ABB RobotStudio station: Robotstudio-car-assembly.rspag

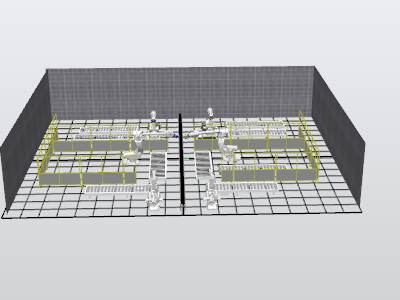
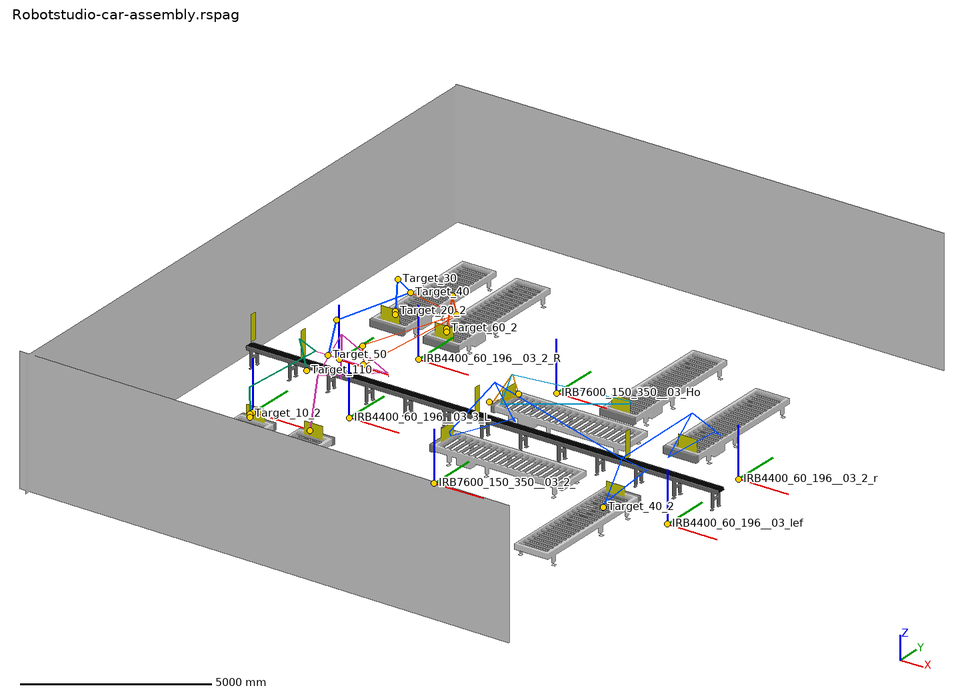
[picture v1: parts stored in the station drawn from their meshes, with robot base, taught points and paths (robot models come from the ABB library and are not in the file)]
--- station ---
Station Project_re_RS (saved by RobotStudio 25.3.11371.0)
Controller Controller29, task T_ROB2: task frame (RAPID world) sits at (6953.35, -1606.5, 0) mm, rotated rx 0 ry 0 rz 180 deg in the station
Controller Controller29, task T_ROB1: task frame (RAPID world) sits at (6953.35, -1606.5, 0) mm, rotated rx 0 ry 0 rz 180 deg in the station
Controller Controller25, task T_ROB2: task frame (RAPID world) sits at (641.16, 3478.05, 0) mm, rotated rx 0 ry 0 rz -90 deg in the station
Controller Controller25, task T_ROB1: task frame (RAPID world) sits at (641.16, 3478.05, 0) mm, rotated rx 0 ry 0 rz -90 deg in the station
Controller Controller23, task T_ROB2: task frame (RAPID world) sits at (-5299.47, 2064.24, 374.5) mm in the station
Controller Controller23, task T_ROB1: task frame (RAPID world) sits at (-5299.47, 2064.24, 374.5) mm in the station
Controller Controller23
  mechanical unit ROB_1: IRB4400_60_196__03_2_Right_Wheel, 6 joints, base frame (0, 0, 0) mm
  mechanical unit TRACK_1: IRBT4004_STD_0_0_3__04_RightWheel, 1 joints, base frame (0, 0, 0) mm
  mechanical unit ROB_2: IRB4400_60_196__03_3_Left_Wheel, 6 joints, base frame (0, 0, 0) mm
  mechanical unit TRACK_2: IRBT4004_STD_0_0_3__04_2_LeftWheel, 1 joints, base frame (-36.16, -3878.12, 0) mm
Controller Controller25
  mechanical unit ROB_1: IRB7600_150_350__03_HoodWind, 6 joints, base frame (358.26, -535.69, 0) mm
  mechanical unit ROB_2: IRB7600_150_350__03_2_Seat, 6 joints, base frame (6589.94, -77.42, 0) mm, rotated rx 0 ry 0 rz 180 deg
Controller Controller29
  mechanical unit ROB_1: IRB4400_60_196__03_leftSide, 6 joints, base frame (0, 0, 0) mm
  mechanical unit ROB_2: IRB4400_60_196__03_2_rightSide, 6 joints, base frame (15.31, -3252.7, 0) mm
Layout (positions relative to the parent item):
  - SmartComponent_Kaross [smart component]
      signals: DI diStartBelt, DI diNewStation, DO doStartBelt, DO dosink, DI diSink
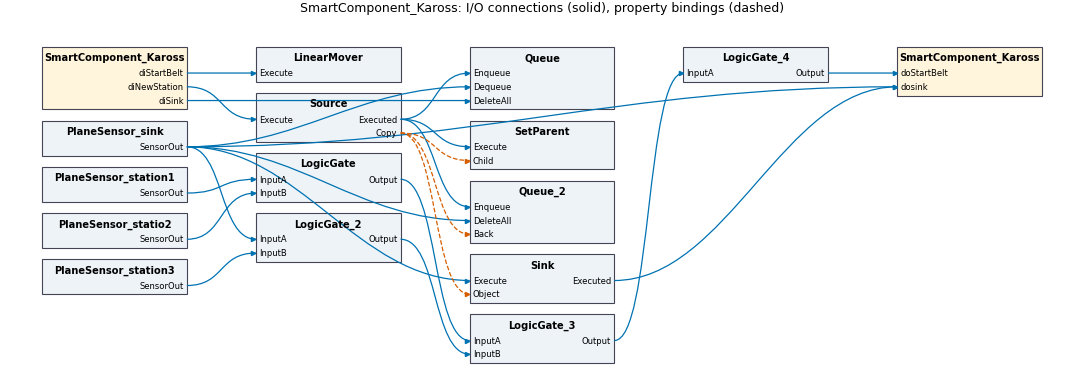
      connections:
        SmartComponent_Kaross.diStartBelt -> LinearMover.Execute
        Source.Executed -> Queue.Enqueue
        PlaneSensor_sink.SensorOut -> Sink.Execute
        PlaneSensor_sink.SensorOut -> Queue.Dequeue
        Source.Executed -> SetParent.Execute
        PlaneSensor_station1.SensorOut -> LogicGate.InputA
        PlaneSensor_statio2.SensorOut -> LogicGate.InputB
        PlaneSensor_sink.SensorOut -> LogicGate_2.InputA
        PlaneSensor_station3.SensorOut -> LogicGate_2.InputB
        LogicGate.Output -> LogicGate_3.InputA
        LogicGate_2.Output -> LogicGate_3.InputB
        LogicGate_3.Output -> LogicGate_4.InputA
        LogicGate_4.Output -> SmartComponent_Kaross.doStartBelt
        SmartComponent_Kaross.diNewStation -> Source.Execute
        Sink.Executed -> SmartComponent_Kaross.dosink
        SmartComponent_Kaross.diSink -> Queue.DeleteAll
        Source.Executed -> Queue_2.Enqueue
        PlaneSensor_sink.SensorOut -> Queue_2.DeleteAll
        PlaneSensor_sink.SensorOut -> SmartComponent_Kaross.dosink
        Source.Copy => SetParent.Child
        Source.Copy => Sink.Object
        Source.Copy => Queue_2.Back
    - Belt Conveyor [part], size 15091 x 400 x 600 mm
    - kaross [part], size 2040 x 1220 x 356.4 mm
    - Source [smart component, from Components\Source.rslib]
        properties: Source=kaross; Copy=(none); Parent=(none); Position=[0 0 0]; Orientation=[0 0 0]; Transient=false; PhysicsBehavior=-1
    - Queue [smart component, from Components\Queue.rslib]
        properties: Back=CAR; Front=(none); Queue=; NumberOfObjects=0
    - LinearMover [smart component, from Components\LinearMover.rslib]
        properties: Object=Queue; Direction=[-1 0 0]; Speed=0.5; Reference=Global; ReferenceObject=(none)
    - PlaneSensor_station1 [smart component, from Components\PlaneSensor.rslib] at (4530.08, -56.57, 1401.52) mm, rotated rx -90 ry 0 rz 90 deg
        properties: Origin=[0 0 0]; Axis1=[0.2 0 0]; Axis2=[0 0.8 0]; Tag=(none); SenseMultiple=false; SensedPart=(none)
      - _sensorPart_ [part], size 200 x 800 x 0 mm
    - PlaneSensor_sink [smart component, from Components\PlaneSensor.rslib] at (-7451.46, 0, 1424.26) mm, rotated rx -90 ry 0 rz 90 deg
        properties: Origin=[0 0 0]; Axis1=[0.2 0 0]; Axis2=[0 0.8 0]; Tag=(none); SenseMultiple=false; SensedPart=(none)
      - _sensorPart_ [part], size 200 x 800 x 0 mm
    - PlaneSensor_statio2 [smart component, from Components\PlaneSensor.rslib] at (-173.15, 0, 622.02) mm, rotated rx 90 ry 0 rz -90 deg
        properties: Origin=[0 0 0]; Axis1=[0.2 0 0]; Axis2=[0 0.8 0]; Tag=(none); SenseMultiple=false; SensedPart=(none)
      - _sensorPart_ [part], size 200 x 800 x 0 mm
    - PlaneSensor_station3 [smart component, from Components\PlaneSensor.rslib] at (-5859.99, 0, 1399.15) mm, rotated rx -90 ry 0 rz 90 deg
        properties: Origin=[0 0 0]; Axis1=[0.2 0 0]; Axis2=[0 0.8 0]; Tag=(none); SenseMultiple=false; SensedPart=(none)
      - _sensorPart_ [part], size 200 x 800 x 0 mm
    - SetParent [smart component, from Components\SetParent.rslib]
        properties: Child=(none); Parent=CAR; KeepTransform=true
    - LogicGate [smart component, from Components\LogicGate.rslib]
        properties: Operator=OR; Delay=0
    - LogicGate_2 [smart component, from Components\LogicGate.rslib]
        properties: Operator=OR; Delay=0
    - LogicGate_3 [smart component, from Components\LogicGate.rslib]
        properties: Operator=OR; Delay=0
    - LogicGate_4 [smart component, from Components\LogicGate.rslib]
        properties: Operator=NOT; Delay=0
    - Queue_2 [smart component, from Components\Queue.rslib]
        properties: Back=(none); Front=(none); Queue=; NumberOfObjects=0
  - IRB4400_60_196__03_2_Right_Wheel [mechanism, from %ABB.RobotStudio.Models.IRB4400%\IRB4400_60_196_G_03.rslib] at (-3551.34, 2064.24, 374.5) mm; joint values [0, 0, 0, 0, 0.5236, 0] (rad or m)
  - IRBT4004_STD_0_0_3__04_RightWheel [mechanism] at (-5694.97, 1504.24, 0) mm; joint values [1.7481] (rad or m)
      links: Base, Link1
  - IRB4400_60_196__03_3_Left_Wheel [mechanism, from %ABB.RobotStudio.Models.IRB4400%\IRB4400_60_196_G_03.rslib] at (-3045.44, -1813.88, 374.5) mm; joint values [0, 0, 0, 0, 0.5236, 0] (rad or m)
  - IRBT4004_STD_0_0_3__04_2_LeftWheel [mechanism] at (-5731.12, -2373.88, 0) mm; joint values [2.2902] (rad or m)
      links: Base, Link1
  - SmartComponent_LeftWheelTool [smart component] at (-2350.09, 2064.24, 2024.5) mm, rotated rx 180 ry 60 rz 180 deg
      signals: DI diGripWheel, DO doGrippedWheel, DI disink
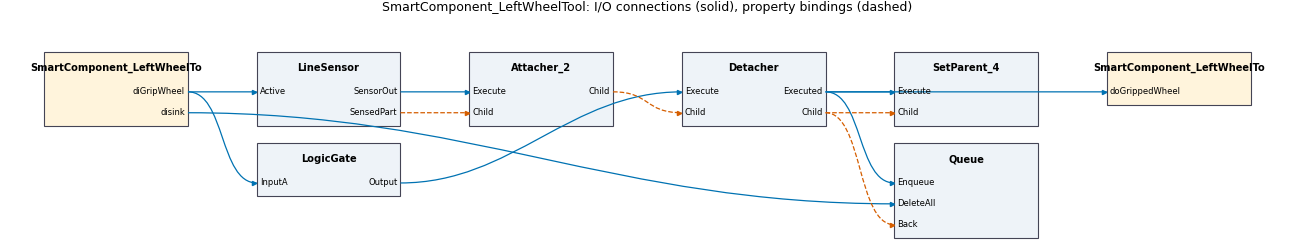
      connections:
        SmartComponent_LeftWheelTool.diGripWheel -> LineSensor.Active
        SmartComponent_LeftWheelTool.diGripWheel -> LogicGate.InputA
        LineSensor.SensorOut -> Attacher_2.Execute
        LogicGate.Output -> Detacher.Execute
        Detacher.Executed -> SmartComponent_LeftWheelTool.doGrippedWheel
        Detacher.Executed -> SetParent_4.Execute
        Detacher.Executed -> Queue.Enqueue
        SmartComponent_LeftWheelTool.disink -> Queue.DeleteAll
        LineSensor.SensedPart => Attacher_2.Child
        Attacher_2.Child => Detacher.Child
        Detacher.Child => SetParent_4.Child
        Detacher.Child => Queue.Back
    - wheeltool [mechanism] at (0, 0, 0) mm
        TCP wheeltool at (0, 0, 20) mm
        links: wheeltool
    - Attacher_2 [smart component, from Components\Attacher.rslib]
        properties: Parent=wheeltool; Flange=0; Child=(none); Mount=false; Offset=[0 0 0]; Orientation=[0 0 0]
    - Detacher [smart component, from Components\Detacher.rslib]
        properties: Child=(none); KeepPosition=true
    - LogicGate [smart component, from Components\LogicGate.rslib]
        properties: Operator=NOT; Delay=0
    - LineSensor [smart component, from Components\LineSensor.rslib] at (104.97, -0.88, 47.26) mm
        properties: Start=[0 0 0]; End=[0 0 0.05]; Length=0.05; Radius=0.00410958904109589; Tag=(none); SenseMultiple=false; SensedPart=(none); SensedPoint=[-4.22472412109375 0.63572021484375 0.5618896484375]
      - _sensorPart_ [part], size 8.2 x 8.2 x 50 mm
    - SetParent_4 [smart component, from Components\SetParent.rslib]
        properties: Child=(none); Parent=CAR; KeepTransform=true
    - Queue [smart component, from Components\Queue.rslib]
        properties: Back=(none); Front=(none); Queue=; NumberOfObjects=0
  - SmartComponent_RightWheelTool [smart component] at (-1844.19, -1813.87, 2024.5) mm, rotated rx -180 ry 60 rz -180 deg
      signals: DI diGripWheel, DO doGrippedWheel, DI disink
      connections:
        SmartComponent_RightWheelTool.diGripWheel -> LineSensor.Active
        SmartComponent_RightWheelTool.diGripWheel -> LogicGate.InputA
        LineSensor.SensorOut -> Attacher_2.Execute
        LogicGate.Output -> Detacher.Execute
        Detacher.Executed -> SmartComponent_RightWheelTool.doGrippedWheel
        Detacher.Executed -> SetParent_5.Execute
        Detacher.Executed -> Queue_3.Enqueue
        SmartComponent_RightWheelTool.disink -> Queue_3.DeleteAll
        LineSensor.SensedPart => Attacher_2.Child
        Attacher_2.Child => Detacher.Child
        Detacher.Child => SetParent_5.Child
        Detacher.Child => Queue_3.Back
    - wheeltool [mechanism] at (0, 0, 0) mm
        TCP wheeltool at (0, 0, 20) mm
        links: wheeltool
    - Attacher_2 [smart component, from Components\Attacher.rslib]
        properties: Parent=wheeltool; Flange=0; Child=(none); Mount=false; Offset=[0 0 0]; Orientation=[0 0 0]
    - Detacher [smart component, from Components\Detacher.rslib]
        properties: Child=(none); KeepPosition=true
    - LogicGate [smart component, from Components\LogicGate.rslib]
        properties: Operator=NOT; Delay=0
    - LineSensor [smart component, from Components\LineSensor.rslib] at (182.92, 28.94, 169.31) mm
        properties: Start=[-0.086602210384922 -3.81423338025044E-07 -0.0499999703769043]; End=[-0.114585975282977 -3.81739185347946E-07 -0.146004704125456]; Length=0.1; Radius=0.00228310502283105; Tag=(none); SenseMultiple=false; SensedPart=(none); SensedPoint=[-4.1956533203125 -0.449598297119141 0.74006982421875]
      - _sensorPart_ [part], size 32.4 x 4.6 x 97.3 mm
    - SetParent_5 [smart component, from Components\SetParent.rslib]
        properties: Child=(none); Parent=CAR; KeepTransform=true
    - Queue_3 [smart component, from Components\Queue.rslib]
        properties: Back=(none); Front=(none); Queue=; NumberOfObjects=0
  - SmartComponent_RightfrontWheelConveyor [smart component] at (-4910.74, 3319.86, 0) mm, rotated rx 0 ry 0 rz 90 deg
      signals: DI DiStartRearWheelCOnveyor
      connections:
        SmartComponent_RightfrontWheelConveyor.DiStartRearWheelCOnveyor -> Source.Execute
        PlaneSensor.SensorOut -> Queue.Dequeue
        Source.Executed -> Queue.Enqueue
        Source.Copy => Queue.Back
    - 950_4000_h2 [part], size 4244 x 1170 x 435 mm
    - Queue [smart component, from Components\Queue.rslib]
        properties: Back=(none); Front=(none); Queue={fd7b7dff-b319-44f7-9117-b8347e8ab7cd};{67428751-7358-4330-9e5c-983121ad5e4f};{f57d0df5-fe45-4d97-8b74-d221833b55af};{56c6505a-fd1b-489a-aa4a-bff5d0e38b36};{77b6cb7b-b71e-4fa1-b8ac-8daa7c661d7c};{7c9591ad-7720-4a29-8a41-6cd58b9ecd19};{fcddd9ad-4e07-40c0-b22b-7d507a136dd0};{d7a43dc1-d6ac-4686-9ac9-cc80a65d254d};{a5e115b4-307d-490d-9473-98725ade6dc6};{a587fca7-a609-44e8-ad7c-b3e0c241758b};{d830a598-c386-40b6-bbb7-414ddccaf421};{461b1b08-72c6-4d72-b9cb-cd15aba64bb5};{e56479b2-e11c-47c7-bcf6-35c12d27192a};{87ffc45d-461f-49e5-a41d-eea24b9ad186};{7c17f912-f0d2-480f-ab99-382f111adc96};{53b25760-ee57-47e1-8360-f256bfaf729e};{619e9f0c-1438-4ff0-a9b2-cfe6a099c667};{804d0500-68f5-4d79-8c34-d375fca0ef9e};{b25e62b0-4662-451b-8aaf-a3910dd8de3a};{166b8770-5aee-437e-91f3-d77d6e0cf809};{fe402c61-951f-47a2-a70e-ae4f84d48686};{c3f4e4fe-14d5-47fb-b26b-3f03b5c19dd2}; NumberOfObjects=0
    - Source [smart component, from Components\Source.rslib]
        properties: Source=frontWheel; Copy=(none); Parent=(none); Position=[0 0 0]; Orientation=[0 0 0]; Transient=false; PhysicsBehavior=-1
    - LinearMover [smart component, from Components\LinearMover.rslib] at (0, 0, 1118.29) mm
        properties: Object=Queue; Direction=[0 -1 0]; Speed=0.5; Reference=Global; ReferenceObject=(none)
    - PlaneSensor [smart component, from Components\PlaneSensor.rslib] at (68.9, 174.35, 837.97) mm, rotated rx 0 ry 90 rz 0 deg
        properties: Origin=[0 0 0]; Axis1=[0.4 0 0]; Axis2=[0 0.6 0]; Tag=(none); SenseMultiple=false; SensedPart=(none)
      - _sensorPart_ [part], size 400 x 600 x 0 mm
  - rearWheel [part], size 399.7 x 400 x 180 mm
  - SmartComponent_LeftfrontWheelConveyor [smart component] at (-5598.22, -3650.57, -183.94) mm, rotated rx 0 ry 0 rz -90 deg
      signals: DI DiStartRightRearWheelCOnveyor
      connections:
        PlaneSensor.SensorOut -> Queue.Dequeue
        Source.Executed -> Queue.Enqueue
        SmartComponent_LeftfrontWheelConveyor.DiStartRightRearWheelCOnveyor -> Source.Execute
        Source.Copy => Queue.Back
    - 950_4000_h2 [part] at (-593.34, 0, 0) mm, size 4244 x 1170 x 435 mm
    - Queue [smart component, from Components\Queue.rslib]
        properties: Back=(none); Front=(none); Queue={7bab526b-e7f3-4f97-a91d-01c49b526e96};{bd76b88b-f630-4995-8fba-bdc71ddf0666};{d1dded0a-8671-4fc3-8d37-267aa8490337};{5deea5c3-a480-4ea7-9b54-bdf3c475bdf6};{955ea6a1-5dc4-422f-a375-dfe26a098746};{ec8ef05a-7591-4b39-a81a-bb7da7deed46};{247e0c03-cbc4-4754-9339-68d3d194897a};{0cf0a9f7-d056-43e1-a56e-a9a3338781c4};{6f5303df-cc14-4586-b84f-762f4a8b9a4f};{31dc02b0-de60-4aa9-8021-4b154c545d33};{a47ea1b2-edb9-4bd1-9507-d2fec89e4b8b};{c3bf3698-6ab2-42cb-8d69-79fb937df227};{779dc5ca-f3d5-4ce3-835a-b32520275891};{6e213d3a-3401-4c3a-8584-7d0b7e865116};{9015acb2-25a2-4553-b97a-6e3350e591a1};{7712fdb7-c615-4efb-b6f8-dc48f9e8acc9};{be5be349-ebb1-4d7f-8bdd-ea2da4429e27};{dc378291-761a-4914-9727-9ab95fa1ad9c};{e7858f16-eb69-476e-96fb-a4ed56d209e4};{72b9bf13-0911-4449-8aa3-f4926b70e8a8};{13c5a77c-64e9-42fc-b696-d95a05be4066};{60331e5b-7cd6-47b6-bf5a-3800f497fbf9};{f650d7cd-82e0-42a7-b45e-2cad3589d1ce};{3e7bd7d4-c306-487b-a1c5-a5dc4588b5fa};{88c07c39-bf5b-4e23-a73f-fb5e2b2d8191};{0decc34c-cdac-4896-b978-958c28f25643};{79729267-b41f-4965-b702-262cb35aaf44};{cb114fb4-7819-4d26-853a-f08010b2a7bf};{a7bd1957-454c-4812-9478-672e2cdcb345};{be25f038-9b73-41fb-8a48-72b7c1c2509f};{30dfbaba-2d50-406d-8718-a595e78b5287};{333c9c72-7684-4034-8313-92e9357a904c};{b128f185-1a74-4133-9f3a-46437fbf5e5e};{388fee6d-961f-4223-bc0a-d61c17e5e143}; NumberOfObjects=0
    - Source [smart component, from Components\Source.rslib]
        properties: Source=frontWheel_2; Copy=(none); Parent=(none); Position=[0 0 0]; Orientation=[0 0 0]; Transient=false; PhysicsBehavior=-1
    - LinearMover [smart component, from Components\LinearMover.rslib] at (0, 0, 1118.29) mm
        properties: Object=Queue; Direction=[0 1 0]; Speed=0.5; Reference=Global; ReferenceObject=(none)
    - PlaneSensor [smart component, from Components\PlaneSensor.rslib] at (-516.51, 174.35, 837.97) mm, rotated rx 0 ry 90 rz 0 deg
        properties: Origin=[0 0 0]; Axis1=[0.4 0 0]; Axis2=[0 0.6 0]; Tag=(none); SenseMultiple=false; SensedPart=(none)
      - _sensorPart_ [part], size 400 x 600 x 0 mm
  - rearWheel_2 [part], size 399.7 x 400 x 180 mm
  - SmartComponent_RightrearWheelConveyor [smart component] at (-3178.8, 3294.07, 0) mm, rotated rx 0 ry 0 rz 90 deg
      signals: DI DiStartLeftFrontWheelCOnveyor
      connections:
        PlaneSensor.SensorOut -> Queue.Dequeue
        Source.Executed -> Queue.Enqueue
        SmartComponent_RightrearWheelConveyor.DiStartLeftFrontWheelCOnveyor -> Source.Execute
        Source.Copy => Queue.Back
    - 950_4000_h2 [part], size 4244 x 1170 x 435 mm
    - Queue [smart component, from Components\Queue.rslib]
        properties: Back=(none); Front=(none); Queue={77faa776-c4b1-45d1-9e5b-038359762285};{a31d55a2-c3cc-456d-a84c-3da71f06c997};{f3487c22-313e-47bd-899e-b4b7b6257dd5};{42bdcfe8-09c7-49d4-9dbf-e1a3af119b64};{ee167c9c-383f-44e9-a683-5fc524fb4b0c};{2eb3e622-42bf-4316-babb-4eaf79ee972c};{61c6edfa-d4dd-4d3c-a615-11f1b465d7c0};{dfefe402-b151-4032-87b4-2dd266781ada};{9fe0b2a1-0ae2-4a62-acc7-1c1a2f093350};{3fa4ad5f-aa0a-4486-92e7-6938df7ae168};{c01374c5-3488-41cb-aa8b-a66ab5a2e7d0};{cebe1a23-2916-499b-8be7-2f12e7de99e4};{dec8808d-e7c3-4b72-94ed-8902570e163a};{143c2350-2b17-4cc7-b77f-2682e3d57473};{a708f5d6-4cb2-40c7-8bbb-bf6ee0d305c4};{565afdcd-3fcb-47df-b43e-8a2b84dba7c1};{8b6458ec-cb0f-4876-9faa-c3b269c4701c};{ca918905-f368-471b-b107-08a5b81300ff};{fb27a522-9416-4fc8-940b-e8c304eeef3e};{642d2391-f722-46f4-8df7-3ed95afff179};{d2453cb7-39b8-4501-b291-1212ce3a701d};{1350be6e-035d-47b1-bfad-abd45f7849d2};{034bca5a-d54d-426a-b0a2-3a655d5b5a22};{493db9ed-35f3-47d8-81b3-40fb8d63b2f8};{3c1a20a6-7b98-4e19-93a2-9cc64df8a6be};{de52d7dc-feaf-4110-bef9-845147e91157}; NumberOfObjects=0
    - Source [smart component, from Components\Source.rslib]
        properties: Source=rearWheel; Copy=(none); Parent=(none); Position=[0 0 0]; Orientation=[0 0 0]; Transient=false; PhysicsBehavior=-1
    - LinearMover [smart component, from Components\LinearMover.rslib] at (0, 0, 1118.29) mm
        properties: Object=Queue; Direction=[0 -1 0]; Speed=0.5; Reference=Global; ReferenceObject=(none)
    - PlaneSensor [smart component, from Components\PlaneSensor.rslib] at (68.9, 174.35, 837.97) mm, rotated rx 0 ry 90 rz 0 deg
        properties: Origin=[0 0 0]; Axis1=[0.4 0 0]; Axis2=[0 0.6 0]; Tag=(none); SenseMultiple=false; SensedPart=(none)
      - _sensorPart_ [part], size 400 x 600 x 0 mm
  - frontWheel [part], size 349 x 350 x 130 mm
  - SmartComponent_LeftrearWheelConveyor [smart component] at (-3634, -3203.27, 0) mm, rotated rx 0 ry 0 rz -90 deg
      signals: DI DiStartRightFrontWheelCOnveyor
      connections:
        PlaneSensor.SensorOut -> Queue.Dequeue
        Source.Executed -> Queue.Enqueue
        SmartComponent_LeftrearWheelConveyor.DiStartRightFrontWheelCOnveyor -> Source.Execute
        Source.Copy => Queue.Back
    - 950_4000_h2 [part], size 4244 x 1170 x 435 mm
    - Queue [smart component, from Components\Queue.rslib]
        properties: Back=(none); Front=(none); Queue={b73c2cab-91c0-4705-8506-9606f316245d};{9eaf44bf-874b-42c6-938f-55b9b2ff61af};{a26c88d9-59a4-4923-9eee-817532e89691};{f43362f0-c841-4eac-b91a-47ef9db6c538};{82b80a5b-797d-4674-b0c3-b733c5cdaa4f};{f3100580-387e-4d05-a987-6845ffbbba7b};{3af67a01-2a3b-4b50-a791-4b1678445dd6};{f4705c2a-f4ee-4ac5-ab5c-836d02fac5b2};{881096ff-7714-419e-979e-2b5f4241d7fd};{ea0002f0-3719-4364-8ee2-2bef2f699958};{451fffa0-3fd4-4854-9cc9-8bc723fda069};{99a6467f-e289-4b56-a678-276a305d6491};{4d66f6b2-efa0-4900-8b93-fbd19e864b79};{bb4fb3fa-ccb6-4199-be74-9ffd31e00806};{dac90289-b8cc-4cb3-a9ea-92585d865125};{860d7759-718d-4ab9-a512-7b287f16d817};{0bdf2866-f8e2-4833-a567-29927e9d811a};{5acf312f-58fc-409c-a6ad-4b71dfd3a6fb};{f45c7ec4-5577-465d-93a4-72ba8a4371ed};{ca2a0b44-0920-4cb2-8538-a4a1e49213c5};{3c09dec7-8001-442d-a323-eafc7ec5860a};{e5d65b8d-1560-4688-aae9-a01a55b4fda5};{78de7aaf-d2f8-458f-a52c-acc46bb5d435};{ae4a09c3-eafd-459d-ac9d-962d8e6b1237};{c78e0534-87c6-4064-8d26-8cfb3fcb1203}; NumberOfObjects=0
    - Source [smart component, from Components\Source.rslib]
        properties: Source=rearWheel_2; Copy=(none); Parent=(none); Position=[0 0 0]; Orientation=[0 0 0]; Transient=false; PhysicsBehavior=-1
    - LinearMover [smart component, from Components\LinearMover.rslib] at (0, 0, 1118.29) mm
        properties: Object=Queue; Direction=[0 1 0]; Speed=0.5; Reference=Global; ReferenceObject=(none)
    - PlaneSensor [smart component, from Components\PlaneSensor.rslib] at (78.09, 174.35, 770.02) mm, rotated rx 0 ry 90 rz 0 deg
        properties: Origin=[0 0 0]; Axis1=[0.4 0 0]; Axis2=[0 0.6 0]; Tag=(none); SenseMultiple=false; SensedPart=(none)
      - _sensorPart_ [part], size 400 x 600 x 0 mm
  - frontWheel_2 [part], size 349 x 350 x 130 mm
  - IRB7600_150_350__03_HoodWind [mechanism, from %ABB.RobotStudio.Models.IRB7600%\IRB7600_150_350_G_03.rslib] at (105.47, 3119.79, 0) mm, rotated rx 0 ry 0 rz -90 deg; joint values [0.2177, 0.0546, -0.0554, -0.3575, 0.5639, 0.416] (rad or m)
  - SmartComponent_1_HoodWind [smart component]
      signals: DI DiStartLeftSide
      connections:
        PlaneSensor.SensorOut -> Queue.Dequeue
        Source.Executed -> Queue.Enqueue
        SmartComponent_1_HoodWind.DiStartLeftSide -> Source.Execute
        Source.Copy => Queue.Back
    - 950_4000_h2 [part] at (-273.12, 900.54, 0) mm, size 4244 x 1170 x 435 mm
    - Queue [smart component, from Components\Queue.rslib] at (-273.12, 900.54, 0) mm
        properties: Back=(none); Front=(none); Queue={74bb35d2-e387-4213-ac07-980f9550285e};{f595998e-2021-4cfe-834f-70741d361f77};{217f4cfc-f555-4b38-8286-b65f35450a09}; NumberOfObjects=0
    - Source [smart component, from Components\Source.rslib] at (-273.12, 900.54, 0) mm
        properties: Source=hood; Copy=(none); Parent=(none); Position=[0 0 0]; Orientation=[0 0 0]; Transient=false; PhysicsBehavior=-1
    - LinearMover [smart component, from Components\LinearMover.rslib] at (-273.12, 900.54, 1118.29) mm
        properties: Object=Queue; Direction=[-1 0 0]; Speed=0.5; Reference=Global; ReferenceObject=(none)
    - PlaneSensor [smart component, from Components\PlaneSensor.rslib] at (-204.22, 1074.88, 805.57) mm, rotated rx 0 ry 90 rz 0 deg
        properties: Origin=[0 0 0]; Axis1=[0.4 0 0]; Axis2=[0 0.6 0]; Tag=(none); SenseMultiple=false; SensedPart=(none)
      - _sensorPart_ [part], size 400 x 600 x 0 mm
  - leftSide [part], size 404.2 x 2000 x 254.9 mm
  - SmartComponent_1_2_seat [smart component] at (-237.73, -1946.18, 0) mm
      signals: DI DiStartRightSide
      connections:
        PlaneSensor.SensorOut -> Queue.Dequeue
        Source.Executed -> Queue.Enqueue
        SmartComponent_1_2_seat.DiStartRightSide -> Source.Execute
        Source.Copy => Queue.Back
    - 950_4000_h2 [part], size 4244 x 1170 x 435 mm
    - Queue [smart component, from Components\Queue.rslib]
        properties: Back=(none); Front=(none); Queue={84b6711d-903e-43bd-bd6e-6b28068a680b};{91bad0f9-4190-4f0c-ba6c-1b84effe9c3a};{ab1b68dd-540d-4fdc-8759-8e6fd8203ddc};{a9fdacad-8ad5-462b-b80d-ac40920b7b78};{c6438745-5e91-45ef-83a0-ab36dacc907c};{3a7d8883-7061-4e26-a8d2-c7ca8f5fbb0c}; NumberOfObjects=0
    - Source [smart component, from Components\Source.rslib]
        properties: Source=seat; Copy=(none); Parent=(none); Position=[0 0 0]; Orientation=[0 0 0]; Transient=false; PhysicsBehavior=-1
    - LinearMover [smart component, from Components\LinearMover.rslib] at (0, 0, 1118.29) mm
        properties: Object=Queue; Direction=[-1 0 0]; Speed=0.5; Reference=Global; ReferenceObject=(none)
    - PlaneSensor [smart component, from Components\PlaneSensor.rslib] at (68.9, 174.35, 837.97) mm, rotated rx 0 ry 90 rz 0 deg
        properties: Origin=[0 0 0]; Axis1=[0.4 0 0]; Axis2=[0 0.6 0]; Tag=(none); SenseMultiple=false; SensedPart=(none)
      - _sensorPart_ [part], size 400 x 600 x 0 mm
  - IRB7600_150_350__03_2_Seat [mechanism, from %ABB.RobotStudio.Models.IRB7600%\IRB7600_150_350_G_03.rslib] at (563.74, -3111.89, 0) mm, rotated rx 0 ry 0 rz 90 deg; joint values [0, 0, 0, 0, 0.5236, 0] (rad or m)
  - rightSide [part], size 404.2 x 2000 x 254.9 mm
  - SmartComponent_1_3_LeftSideTool [smart component] at (5752.11, -1606.5, 1650) mm, rotated rx -180 ry 60 rz 0 deg
      signals: DI diGripSide, DO doGrippedSide, DI disink
      connections:
        SmartComponent_1_3_LeftSideTool.diGripSide -> LineSensor.Active
        SmartComponent_1_3_LeftSideTool.diGripSide -> LogicGate.InputA
        LogicGate.Output -> Detacher.Execute
        LineSensor.SensorOut -> Attacher.Execute
        Detacher.Executed -> SmartComponent_1_3_LeftSideTool.doGrippedSide
        Detacher.Executed -> SetParent_6.Execute
        Detacher.Executed -> Queue_2.Enqueue
        SmartComponent_1_3_LeftSideTool.disink -> Queue_2.DeleteAll
        LineSensor.SensedPart => Attacher.Child
        Attacher.Child => Detacher.Child
        Detacher.Child => SetParent_6.Child
        Detacher.Child => Queue_2.Back
    - LeftsideTool [mechanism, from Libraries\sideTool.rslib] at (0, 0, 0) mm
    - Attacher [smart component, from Components\Attacher.rslib]
        properties: Parent=LeftsideTool; Flange=0; Child=(none); Mount=false; Offset=[0 0 0]; Orientation=[0 0 0]
    - Detacher [smart component, from Components\Detacher.rslib]
        properties: Child=(none); KeepPosition=true
    - LogicGate [smart component, from Components\LogicGate.rslib]
        properties: Operator=NOT; Delay=0
    - LineSensor [smart component, from Components\LineSensor.rslib] at (-28.91, 89.22, 221.77) mm, rotated rx -90 ry 0 rz 15.45 deg
        properties: Start=[0 0 0]; End=[0 0 0.02]; Length=0.02; Radius=0.00228310502283105; Tag=(none); SenseMultiple=false; SensedPart=(none); SensedPoint=[5.52296875 -0.51899755859375 0.724073852539063]
      - _sensorPart_ [part], size 4.6 x 4.6 x 20 mm
    - SetParent_6 [smart component, from Components\SetParent.rslib]
        properties: Child=(none); Parent=CAR; KeepTransform=true
    - Queue_2 [smart component, from Components\Queue.rslib]
        properties: Back=(none); Front=(none); Queue=; NumberOfObjects=0
  - SmartComponent_1_4_RightSideTool [smart component] at (5736.8, 1646.21, 1650) mm, rotated rx -180 ry 60 rz 0 deg
      signals: DI diGripSide, DO doGrippedSide, DI disink
      connections:
        SmartComponent_1_4_RightSideTool.diGripSide -> LineSensor.Active
        SmartComponent_1_4_RightSideTool.diGripSide -> LogicGate.InputA
        LogicGate.Output -> Detacher.Execute
        LineSensor.SensorOut -> Attacher.Execute
        Detacher.Executed -> SmartComponent_1_4_RightSideTool.doGrippedSide
        Detacher.Executed -> SetParent_3.Execute
        Detacher.Executed -> Queue_4.Enqueue
        SmartComponent_1_4_RightSideTool.disink -> Queue_4.DeleteAll
        LineSensor.SensedPart => Attacher.Child
        Attacher.Child => Detacher.Child
        Detacher.Child => SetParent_3.Child
        Detacher.Child => Queue_4.Back
    - RightsideTool [mechanism, from Libraries\sideTool.rslib] at (0, 0, 0) mm
    - Attacher [smart component, from Components\Attacher.rslib]
        properties: Parent=RightsideTool; Flange=0; Child=(none); Mount=false; Offset=[0 0 0]; Orientation=[0 0 0]
    - Detacher [smart component, from Components\Detacher.rslib]
        properties: Child=(none); KeepPosition=true
    - LogicGate [smart component, from Components\LogicGate.rslib]
        properties: Operator=NOT; Delay=0
    - LineSensor [smart component, from Components\LineSensor.rslib] at (-28.91, 99.22, 221.77) mm, rotated rx -90 ry 0 rz 15.45 deg
        properties: Start=[0 0 0]; End=[0 0 0.02]; Length=0.02; Radius=0.00228310502283105; Tag=(none); SenseMultiple=false; SensedPart=(none); SensedPoint=[5.47422802734375 0.53570556640625 0.673378540039063]
      - _sensorPart_ [part], size 4.6 x 4.6 x 20 mm
    - SetParent_3 [smart component, from Components\SetParent.rslib]
        properties: Child=(none); Parent=CAR; KeepTransform=true
    - Queue_4 [smart component, from Components\Queue.rslib]
        properties: Back=(none); Front=(none); Queue=; NumberOfObjects=0
  - Fence_2500 [graphiccomponentgroup, from Equipment\Fence_2500.rslib] at (-1146.76, 872.76, 0) mm
    - Body 1 [part, from Equipment\Fence_2500.rslib]
    - Body 2 [part, from Equipment\Fence_2500.rslib]
  - Fence_2500_2 [graphiccomponentgroup, from Equipment\Fence_2500.rslib] at (-1143.54, 3289.51, 0) mm
    - Body 1 [part, from Equipment\Fence_2500.rslib]
    - Body 2 [part, from Equipment\Fence_2500.rslib]
  - Fence_2500_3 [graphiccomponentgroup, from Equipment\Fence_2500.rslib] at (-1139.03, 5802.85, 0) mm
    - Body 1 [part, from Equipment\Fence_2500.rslib]
    - Body 2 [part, from Equipment\Fence_2500.rslib]
  - Fence_2500_4 [graphiccomponentgroup, from Equipment\Fence_2500.rslib] at (-1267.52, 8287.94, 0) mm, rotated rx 0 ry 0 rz 90 deg
    - Body 1 [part, from Equipment\Fence_2500.rslib]
    - Body 2 [part, from Equipment\Fence_2500.rslib]
  - Fence_2500_5 [graphiccomponentgroup, from Equipment\Fence_2500.rslib] at (-1212.38, -3321.71, 0) mm
    - Body 1 [part, from Equipment\Fence_2500.rslib]
    - Body 2 [part, from Equipment\Fence_2500.rslib]
  - Fence_2500_6 [graphiccomponentgroup, from Equipment\Fence_2500.rslib] at (-1190.89, -5888.84, 0) mm
    - Body 1 [part, from Equipment\Fence_2500.rslib]
    - Body 2 [part, from Equipment\Fence_2500.rslib]
  - Fence_2500_7 [graphiccomponentgroup, from Equipment\Fence_2500.rslib] at (-1188.54, -8426.52, 0) mm
    - Body 1 [part, from Equipment\Fence_2500.rslib]
    - Body 2 [part, from Equipment\Fence_2500.rslib]
  - Fence_2500_8 [graphiccomponentgroup, from Equipment\Fence_2500.rslib] at (-3671.96, -8518.49, 0) mm, rotated rx 0 ry 0 rz -90 deg
    - Body 1 [part, from Equipment\Fence_2500.rslib]
    - Body 2 [part, from Equipment\Fence_2500.rslib]
  - Fence_2500_9 [graphiccomponentgroup, from Equipment\Fence_2500.rslib] at (-1099.44, -8515, 0) mm, rotated rx 0 ry 0 rz -90 deg
    - Body 1 [part, from Equipment\Fence_2500.rslib]
    - Body 2 [part, from Equipment\Fence_2500.rslib]
  - Fence_2500_10 [graphiccomponentgroup, from Equipment\Fence_2500.rslib] at (1428.44, -8518.13, 0) mm, rotated rx 0 ry 0 rz -90 deg
    - Body 1 [part, from Equipment\Fence_2500.rslib]
    - Body 2 [part, from Equipment\Fence_2500.rslib]
  - Fence_2500_11 [graphiccomponentgroup, from Equipment\Fence_2500.rslib] at (4053.25, -8545.36, 0) mm
    - Body 1 [part, from Equipment\Fence_2500.rslib]
    - Body 2 [part, from Equipment\Fence_2500.rslib]
  - Fence_2500_12 [graphiccomponentgroup, from Equipment\Fence_2500.rslib] at (4067.94, -5982.97, 0) mm
    - Body 1 [part, from Equipment\Fence_2500.rslib]
    - Body 2 [part, from Equipment\Fence_2500.rslib]
  - Fence_740 [graphiccomponentgroup, from Equipment\Fence_740.rslib] at (4057.72, -3450.5, 0) mm
    - Body 1 [part, from Equipment\Fence_740.rslib]
    - Body 2 [part, from Equipment\Fence_740.rslib]
  - Fence_2500_13 [graphiccomponentgroup, from Equipment\Fence_2500.rslib] at (-1042.72, 8251.25, 0) mm, rotated rx 0 ry 0 rz -90 deg
    - Body 1 [part, from Equipment\Fence_2500.rslib]
    - Body 2 [part, from Equipment\Fence_2500.rslib]
  - Fence_2500_14 [graphiccomponentgroup, from Equipment\Fence_2500.rslib] at (1536.21, 8249.03, 0) mm, rotated rx 0 ry 0 rz -90 deg
    - Body 1 [part, from Equipment\Fence_2500.rslib]
    - Body 2 [part, from Equipment\Fence_2500.rslib]
  - Fence_2500_15 [graphiccomponentgroup, from Equipment\Fence_2500.rslib] at (3963.26, 5688, 0) mm
    - Body 1 [part, from Equipment\Fence_2500.rslib]
    - Body 2 [part, from Equipment\Fence_2500.rslib]
  - Fence_2500_16 [graphiccomponentgroup, from Equipment\Fence_2500.rslib] at (3945.06, 3141.67, 0) mm
    - Body 1 [part, from Equipment\Fence_2500.rslib]
    - Body 2 [part, from Equipment\Fence_2500.rslib]
  - Fence_740_2 [graphiccomponentgroup, from Equipment\Fence_740.rslib] at (3948.81, 2383.52, 0) mm
    - Body 1 [part, from Equipment\Fence_740.rslib]
    - Body 2 [part, from Equipment\Fence_740.rslib]
  - Wall [part] at (0, 251.06, 0) mm, size 45.8 x 19721 x 4000 mm
  - Wall [part] at (0, 0, 0) mm, rotated rx 0 ry 0 rz -1.56 deg, size 15766.5 x 221.2 x 4000 mm
  - Wall [part], size 15546.7 x 39 x 4000 mm
  - seat [part], size 229.1 x 800 x 268.8 mm
  - SmartComponent_1_LeftSide [smart component]
      signals: DI DiStartSeat
      connections:
        PlaneSensor.SensorOut -> Queue.Dequeue
        Source.Executed -> Queue.Enqueue
        SmartComponent_1_LeftSide.DiStartSeat -> Source.Execute
        Source.Copy => Queue.Back
    - 950_4000_h2 [part] at (4950.81, -1520.95, 36.4) mm, rotated rx 0 ry 0 rz -90 deg, size 4244 x 1170 x 435 mm
    - Queue [smart component, from Components\Queue.rslib] at (4801.93, -2052.57, 490.52) mm, rotated rx 0 ry 0 rz -90 deg
        properties: Back=(none); Front=(none); Queue={07430233-d3b7-49fd-b9bd-74eda819d421};{a4a4c974-1ee6-4836-868e-efa0c6c08741};{9d930d86-49a8-44e2-90cc-b3aba404a9c0};{65873131-94db-4b90-acdc-57ebd6d7f0b3};{72c35522-4887-4d30-aa15-f0af1a6e0ab9}; NumberOfObjects=0
    - Source [smart component, from Components\Source.rslib] at (4801.93, -2052.57, 490.52) mm, rotated rx 0 ry 0 rz -90 deg
        properties: Source=leftSide; Copy=(none); Parent=(none); Position=[0 0 0]; Orientation=[0 0 0]; Transient=false; PhysicsBehavior=-1
    - LinearMover [smart component, from Components\LinearMover.rslib] at (4801.93, -2052.57, 1608.81) mm, rotated rx 0 ry 0 rz -90 deg
        properties: Object=Queue; Direction=[0 1 0]; Speed=0.5; Reference=Global; ReferenceObject=(none)
    - PlaneSensor [smart component, from Components\PlaneSensor.rslib] at (4976.27, -1598.09, 709.94) mm, rotated rx 0 ry 90 rz -90 deg
        properties: Origin=[0 0 0]; Axis1=[0.4 0 0]; Axis2=[0 0.6 0]; Tag=(none); SenseMultiple=false; SensedPart=(none)
      - _sensorPart_ [part], size 400 x 600 x 0 mm
  - IRB4400_60_196__03_leftSide [mechanism, from %ABB.RobotStudio.Models.IRB4400%\IRB4400_60_196_G_03.rslib] at (6953.35, -1606.5, 0) mm, rotated rx 0 ry 0 rz 180 deg; joint values [0, 0, 0, 0, 0.5236, 0] (rad or m)
  - IRB4400_60_196__03_2_rightSide [mechanism, from %ABB.RobotStudio.Models.IRB4400%\IRB4400_60_196_G_03.rslib] at (6938.04, 1646.21, 0) mm, rotated rx 0 ry 0 rz 180 deg; joint values [0, 0, 0, 0, 0.5236, 0] (rad or m)
  - SmartComponent_1_RightSIde [smart component]
      signals: DI DiStartHood
      connections:
        PlaneSensor.SensorOut -> Queue.Dequeue
        Source.Executed -> Queue.Enqueue
        SmartComponent_1_RightSIde.DiStartHood -> Source.Execute
        Source.Copy => Queue.Back
    - 950_4000_h2 [part] at (5702.88, 1509.58, 0) mm, rotated rx 0 ry 0 rz 90 deg, size 4244 x 1170 x 435 mm
    - Queue [smart component, from Components\Queue.rslib] at (5702.88, 2543.01, 0) mm, rotated rx 0 ry 0 rz 90 deg
        properties: Back=(none); Front=(none); Queue={b0d650cb-51c0-420a-93d1-b0f000a169be};{f51db09f-93e1-4074-b69a-a068383e1127};{9c0fb3bf-1296-4a84-bae8-93f6a30a3feb}; NumberOfObjects=0
    - Source [smart component, from Components\Source.rslib] at (5702.88, 2543.01, 0) mm, rotated rx 0 ry 0 rz 90 deg
        properties: Source=rightSide; Copy=(none); Parent=(none); Position=[0 0 0]; Orientation=[0 0 0]; Transient=false; PhysicsBehavior=-1
    - LinearMover [smart component, from Components\LinearMover.rslib] at (5702.88, 2543.01, 1118.29) mm, rotated rx 0 ry 0 rz 90 deg
        properties: Object=Queue; Direction=[0 -1 0]; Speed=0.5; Reference=Global; ReferenceObject=(none)
    - PlaneSensor [smart component, from Components\PlaneSensor.rslib] at (5636.12, 1608.97, 816.22) mm, rotated rx 0 ry 90 rz 90 deg
        properties: Origin=[0 0 0]; Axis1=[0.4 0 0]; Axis2=[0 0.6 0]; Tag=(none); SenseMultiple=false; SensedPart=(none)
      - _sensorPart_ [part], size 400 x 600 x 0 mm
  - hood [part], size 601.9 x 493.3 x 5 mm
  - SmartComponent_1_3_SeatTool [smart component] at (563.74, -473.38, 1895) mm, rotated rx 180 ry 60 rz -90 deg
      signals: DI diGripseatTool, DO doGrippedseatTool, DI disink
      connections:
        SmartComponent_1_3_SeatTool.diGripseatTool -> LineSensor.Active
        SmartComponent_1_3_SeatTool.diGripseatTool -> LogicGate.InputA
        LineSensor.SensorOut -> Attacher_2.Execute
        LogicGate.Output -> Detacher.Execute
        Detacher.Executed -> SmartComponent_1_3_SeatTool.doGrippedseatTool
        Detacher.Executed -> SetParent.Execute
        Detacher.Executed -> Queue_5.Enqueue
        SmartComponent_1_3_SeatTool.disink -> Queue_5.DeleteAll
        LineSensor.SensedPart => Attacher_2.Child
        Attacher_2.Child => Detacher.Child
        Detacher.Child => SetParent.Child
        Detacher.Child => Queue_5.Back
    - seatTool [mechanism] at (0, 0, 0) mm
        TCP seatTool at (-5.4, 0, 164.64) mm, rotated rx 0 ry -3.73 rz 0 deg
        links: seatTool
    - Attacher_2 [smart component, from Components\Attacher.rslib]
        properties: Parent=seatTool; Flange=0; Child=(none); Mount=false; Offset=[0 0 0]; Orientation=[0 0 0]
    - Detacher [smart component, from Components\Detacher.rslib]
        properties: Child=(none); KeepPosition=true
    - LogicGate [smart component, from Components\LogicGate.rslib]
        properties: Operator=NOT; Delay=0
    - LineSensor [smart component, from Components\LineSensor.rslib] at (0, 0, 167.13) mm
        properties: Start=[0 0 0]; End=[0 0 0.1]; Length=0.1; Radius=0.00228310502283105; Tag=(none); SenseMultiple=false; SensedPart=(none); SensedPoint=[0.948279541015625 0.0129561767578125 0.638018676757813]
      - _sensorPart_ [part], size 4.6 x 4.6 x 100 mm
    - SetParent [smart component, from Components\SetParent.rslib]
        properties: Child=(none); Parent=CAR; KeepTransform=true
    - Queue_5 [smart component, from Components\Queue.rslib]
        properties: Back=(none); Front=(none); Queue=; NumberOfObjects=0
  - SmartComponent_1_4_HoodTool [smart component] at (641.16, 481.28, 1895) mm, rotated rx 180 ry 60 rz 90 deg
      signals: DI diGriphoodWind, DO doGrippedhoodWind, DI disink
      connections:
        SmartComponent_1_4_HoodTool.diGriphoodWind -> LineSensor.Active
        SmartComponent_1_4_HoodTool.diGriphoodWind -> LogicGate.InputA
        LineSensor.SensorOut -> Attacher.Execute
        LogicGate.Output -> Detacher.Execute
        Detacher.Executed -> SmartComponent_1_4_HoodTool.doGrippedhoodWind
        Detacher.Executed -> SetParent_2.Execute
        Detacher.Executed -> Queue_6.Enqueue
        SmartComponent_1_4_HoodTool.disink -> Queue_6.DeleteAll
        LineSensor.SensedPart => Attacher.Child
        Attacher.Child => Detacher.Child
        Detacher.Child => SetParent_2.Child
        Detacher.Child => Queue_6.Back
    - hoodWindTool [mechanism] at (0, 0, 0) mm
        TCP hoodWindTool at (0, 0, 160) mm
        links: hoodWindTool
    - Attacher [smart component, from Components\Attacher.rslib]
        properties: Parent=hoodWindTool; Flange=0; Child=(none); Mount=false; Offset=[0 0 0]; Orientation=[0 0 0]
    - Detacher [smart component, from Components\Detacher.rslib]
        properties: Child=(none); KeepPosition=true
    - LineSensor [smart component, from Components\LineSensor.rslib] at (0, 0, 167.2) mm
        properties: Start=[0 0 0]; End=[0 0 0.1]; Length=0.1; Radius=0.00228310502283105; Tag=(none); SenseMultiple=false; SensedPart=(none); SensedPoint=[0.530458312988281 0.0041767578125 1.02734362792969]
      - _sensorPart_ [part], size 4.6 x 4.6 x 100 mm
    - LogicGate [smart component, from Components\LogicGate.rslib]
        properties: Operator=NOT; Delay=0
    - SetParent_2 [smart component, from Components\SetParent.rslib]
        properties: Child=(none); Parent=CAR; KeepTransform=true
    - Queue_6 [smart component, from Components\Queue.rslib]
        properties: Back=(none); Front=(none); Queue=; NumberOfObjects=0
  - SmartComponent_windsheild [smart component]
      signals: DI DiStartRearWheelCOnveyor
      connections:
        SmartComponent_windsheild.DiStartRearWheelCOnveyor -> Source.Execute
        PlaneSensor.SensorOut -> Queue.Dequeue
        Source.Executed -> Queue.Enqueue
        Source.Copy => Queue.Back
    - 950_4000_h2 [part] at (3057.68, 2432.86, 0) mm, rotated rx 0 ry 0 rz 90 deg, size 4244 x 1170 x 435 mm
    - Queue [smart component, from Components\Queue.rslib] at (3057.68, 2432.86, 0) mm, rotated rx 0 ry 0 rz 90 deg
        properties: Back=(none); Front=(none); Queue={e9447ad6-d9a3-4a92-bb8d-c389303e7b55};{73bab88b-d860-4cba-8244-0688a56d0f8c};{24ee4f5a-f29f-4277-82d5-eca10cdc3600};{8fe8e95f-5031-4424-8299-9bb07082b79b}; NumberOfObjects=0
    - Source [smart component, from Components\Source.rslib] at (3057.68, 2432.86, 0) mm, rotated rx 0 ry 0 rz 90 deg
        properties: Source=windshield_2; Copy=(none); Parent=(none); Position=[0 0 0]; Orientation=[0 0 0]; Transient=false; PhysicsBehavior=-1
    - LinearMover [smart component, from Components\LinearMover.rslib] at (3057.68, 2432.86, 1118.29) mm, rotated rx 0 ry 0 rz 90 deg
        properties: Object=Queue; Direction=[0 -1 0]; Speed=0.5; Reference=Global; ReferenceObject=(none)
    - PlaneSensor [smart component, from Components\PlaneSensor.rslib] at (2883.33, 2501.76, 837.97) mm, rotated rx 0 ry 90 rz 90 deg
        properties: Origin=[0 0 0]; Axis1=[0.4 0 0]; Axis2=[0 0.6 0]; Tag=(none); SenseMultiple=false; SensedPart=(none)
      - _sensorPart_ [part], size 400 x 600 x 0 mm
  - windshield_2 [part], size 320 x 765.6 x 5 mm
  - CAR [graphiccomponentgroup] at (-178524, 0, 0) mm
Attachment: IRB4400_60_196__03_2_Right_Wheel is attached to IRBT4004_STD_0_0_3__04_RightWheel / Link1
Attachment: IRB4400_60_196__03_3_Left_Wheel is attached to IRBT4004_STD_0_0_3__04_2_LeftWheel / Link1
Attachment: SmartComponent_LeftWheelTool is attached to IRB4400_60_196__03_2_Right_Wheel / Link6
Attachment: SmartComponent_1_4_HoodTool is attached to IRB7600_150_350__03_HoodWind / Link6
Attachment: SmartComponent_1_3_SeatTool is attached to IRB7600_150_350__03_2_Seat / Link6
Attachment: SmartComponent_1_3_LeftSideTool is attached to IRB4400_60_196__03_leftSide / Link6
Attachment: SmartComponent_1_4_RightSideTool is attached to IRB4400_60_196__03_2_rightSide / Link6
Attachment: SmartComponent_RightWheelTool is attached to IRB4400_60_196__03_3_Left_Wheel / Link6
Station signals: DI diStartProgram, DI distart
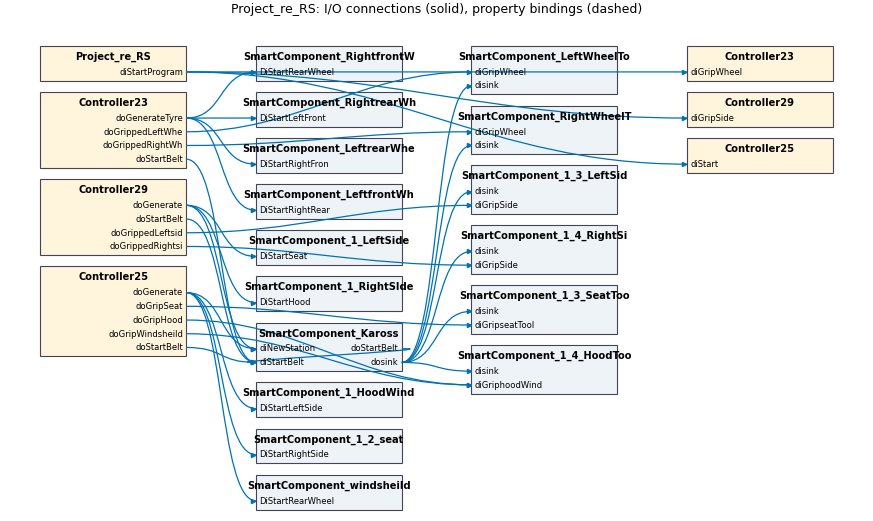
Station logic (signal -> signal, property => property):
  Project_re_RS.diStartProgram -> Controller23.diGripWheel
  Controller23.doGenerateTyre -> SmartComponent_RightfrontWheelConveyor.DiStartRearWheelCOnveyor
  Controller23.doGrippedLeftWheel -> SmartComponent_LeftWheelTool.diGripWheel
  Controller23.doGrippedRightWheel -> SmartComponent_RightWheelTool.diGripWheel
  Controller23.doGenerateTyre -> SmartComponent_RightrearWheelConveyor.DiStartLeftFrontWheelCOnveyor
  Controller23.doGenerateTyre -> SmartComponent_LeftrearWheelConveyor.DiStartRightFrontWheelCOnveyor
  Controller23.doGenerateTyre -> SmartComponent_LeftfrontWheelConveyor.DiStartRightRearWheelCOnveyor
  Controller29.doGenerate -> SmartComponent_Kaross.diNewStation
  Controller29.doStartBelt -> SmartComponent_Kaross.diStartBelt
  SmartComponent_Kaross.doStartBelt -> SmartComponent_Kaross.diStartBelt
  SmartComponent_Kaross.dosink -> SmartComponent_LeftWheelTool.disink
  SmartComponent_Kaross.dosink -> SmartComponent_RightWheelTool.disink
  SmartComponent_Kaross.dosink -> SmartComponent_1_3_LeftSideTool.disink
  SmartComponent_Kaross.dosink -> SmartComponent_1_3_SeatTool.disink
  SmartComponent_Kaross.dosink -> SmartComponent_1_4_HoodTool.disink
  Project_re_RS.diStartProgram -> Controller29.diGripSide
  Controller29.doGrippedLeftside -> SmartComponent_1_3_LeftSideTool.diGripSide
  Controller29.doGenerate -> SmartComponent_1_LeftSide.DiStartSeat
  Controller29.doGenerate -> SmartComponent_1_RightSIde.DiStartHood
  SmartComponent_Kaross.dosink -> SmartComponent_1_4_RightSideTool.disink
  Controller29.doGrippedRightside -> SmartComponent_1_4_RightSideTool.diGripSide
  Project_re_RS.diStartProgram -> Controller25.diStart
  Controller25.doGenerate -> SmartComponent_Kaross.diNewStation
  Controller25.doGripSeat -> SmartComponent_1_3_SeatTool.diGripseatTool
  Controller25.doGenerate -> SmartComponent_1_HoodWind.DiStartLeftSide
  Controller25.doGenerate -> SmartComponent_1_2_seat.DiStartRightSide
  Controller25.doGenerate -> SmartComponent_windsheild.DiStartRearWheelCOnveyor
  Controller25.doGripHood -> SmartComponent_1_4_HoodTool.diGriphoodWind
  Controller25.doGripWindsheild -> SmartComponent_1_4_HoodTool.diGriphoodWind
  Controller25.doStartBelt -> SmartComponent_Kaross.diStartBelt
  Controller23.doStartBelt -> SmartComponent_Kaross.diStartBelt

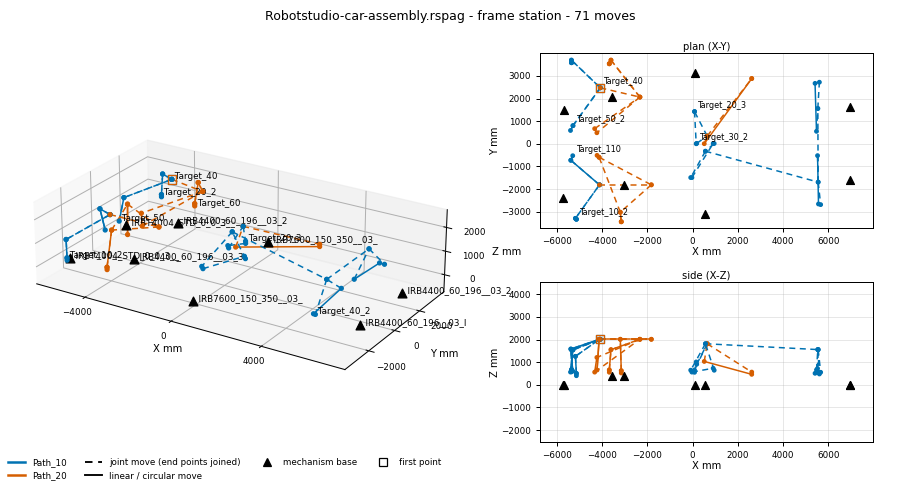
[picture p0: tool path of Robotstudio-car-assembly.rspag in frame station, 71 of 71 moves have a stored position in this frame; points joined in program order, loops and branches not executed]
--- Backups/Controller23/RAPID/TASK1/PROGMOD/CalibData.mod ---
MODULE CalibData
    PERS tooldata wheeltool_left:=[TRUE,[[0,0,20],[1,0,0,0]],[1,[0,0,1],[1,0,0,0],0,0,0]];
    TASK PERS wobjdata Workobject_1:=[FALSE,TRUE,"",[[-621.267,1131.62,60.5],[0,0.707107,0.707107,0]],[[0,0,0],[1,0,0,0]]];
ENDMODULE

--- Backups/Controller23/RAPID/TASK1/PROGMOD/Module1.mod ---
MODULE Module1
    CONST robtarget Target_40:=[[-723.199878422,1839.83102347,-1579.5],[0.612372436,-0.353553391,-0.353553391,-0.612372436],[0,-1,0,0],[0,9E+09,9E+09,9E+09,9E+09,9E+09]];
    CONST robtarget Target_30:=[[500.87367895,562.975012033,-1118.987834532],[0.662080597,0.256994793,0.239274352,0.662080618],[1,-1,-1,0],[0,9E+09,9E+09,9E+09,9E+09,9E+09]];
    CONST robtarget Target_20_2:=[[386.61,567.055,-241.416],[0.707106781,0,0,0.707106781],[1,0,-1,0],[0,9E+09,9E+09,9E+09,9E+09,9E+09]];
    CONST robtarget Target_20:=[[386.61,567.055,-141.416],[0.707106781,0,0,0.707106781],[0,0,0,0],[0,9E+09,9E+09,9E+09,9E+09,9E+09]];
    CONST robtarget Target_50:=[[-2607.141607902,522.859157526,-130.278],[0.5,-0.5,-0.5,0.5],[-1,0,0,0],[0,9E+09,9E+09,9E+09,9E+09,9E+09]];
    CONST robtarget Target_80:=[[-1131.619983054,3587.961864591,-1579.5],[0.612372436,-0.353553391,-0.353553391,-0.612372436],[-1,0,-1,0],[1748.130841122,9E+09,9E+09,9E+09,9E+09,9E+09]];
    CONST robtarget Target_70:=[[500.874033397,2311.10564668,-1118.988029665],[0.662080641,0.256994894,0.239274453,0.662080498],[1,-1,-1,0],[1748.130841122,9E+09,9E+09,9E+09,9E+09,9E+09]];
    CONST robtarget Target_60_2:=[[340.332,2236.709,-222.21],[0.707106781,0,0,0.707106781],[1,0,-1,0],[1748.130841122,9E+09,9E+09,9E+09,9E+09,9E+09]];
    CONST robtarget Target_60:=[[340.332,2236.709,-122.21],[0.707106781,0,0,0.707106781],[1,0,-1,0],[1748.130841122,9E+09,9E+09,9E+09,9E+09,9E+09]];
    CONST robtarget Target_100:=[[-2708.293723211,1687.113860643,-776.398297742],[0.969071906,0.124507933,-0.188250825,-0.099795003],[-2,-1,-1,0],[1206.074766355,9E+09,9E+09,9E+09,9E+09,9E+09]];
    CONST robtarget Target_90:=[[-2526.74990942,1591.043258602,-127.768488614],[0.5,-0.5,-0.5,0.5],[-2,1,-1,0],[1748.130841122,9E+09,9E+09,9E+09,9E+09,9E+09]];
    CONST robtarget Target_50_2:=[[-2394.597661695,631.947,-1108.559888271],[0.5,-0.5,-0.5,0.5],[-1,0,0,0],[0,9E+09,9E+09,9E+09,9E+09,9E+09]];
    CONST robtarget Target_90_2:=[[-2568.922,1811.436,-195.278],[0.5,-0.5,-0.5,0.5],[-2,-1,-3,0],[1748.130841122,9E+09,9E+09,9E+09,9E+09,9E+09]];
    !***********************************************************
    !
    ! Module:  Module1
    !
    ! Description:
    !   <Insert description here>
    !
    ! Author: tmoun
    !
    ! Version: 1.0
    !
    !***********************************************************


    !***********************************************************
    !
    ! Procedure main
    !
    !   This is the entry point of your program
    !
    !***********************************************************
    PROC main()
        !Add your code here
        SetDo doGrippedLeftWheel, 0;
        WaitDI diGripWheel,0;
        SetDO doGenerateTyre, 1;
        SetDO doGenerateTyre, 0;
        SetDO doStartBelt, 0;
        WaitTime 10;
        Path_10;
        Path_20;
    ENDPROC
    PROC Path_10()
        SetDO doStartBelt, 0;
        WaitTime 35;
        MoveJ Target_40,v1000,z0,wheeltool_left\WObj:=Workobject_1;
        MoveJ Target_30,v1000,z0,wheeltool_left\WObj:=Workobject_1;
        MoveJ Target_20_2,v1000,z0,wheeltool_left\WObj:=Workobject_1;
        MoveL Target_20,v1000,fine,wheeltool_left\WObj:=Workobject_1;
        WaitTime 2;
        SetDO doGrippedLeftWheel, 1;
        WaitTime 1;
        MoveL Target_20_2,v1000,fine,wheeltool_left\WObj:=Workobject_1;
        MoveJ Target_30,v1000,z0,wheeltool_left\WObj:=Workobject_1;
        MoveJ Target_40,v1000,z0,wheeltool_left\WObj:=Workobject_1;
        MoveJ Target_50_2,v1000,z0,wheeltool_left\WObj:=Workobject_1;
        MoveL Target_50,v1000,fine,wheeltool_left\WObj:=Workobject_1;
        WaitTime 1;
        SetDO doGrippedLeftWheel, 0;
        WaitTime 1;
        MoveJ Target_50_2,v1000,z0,wheeltool_left\WObj:=Workobject_1;
        MoveJ Target_40,v1000,fine,wheeltool_left\WObj:=Workobject_1;
    ENDPROC
    PROC Path_20()
        MoveJ Target_40,v1000,z0,wheeltool_left\WObj:=Workobject_1;
        MoveJ Target_80,v1000,z0,wheeltool_left\WObj:=Workobject_1;
        MoveJ Target_70,v1000,z0,wheeltool_left\WObj:=Workobject_1;
        MoveL Target_60_2,v1000,fine,wheeltool_left\WObj:=Workobject_1;
        MoveL Target_60,v1000,fine,wheeltool_left\WObj:=Workobject_1;
        WaitTime 1;
        SetDO doGrippedLeftWheel, 1;
        WaitTime 1;
        MoveJ Target_60_2,v1000,fine,wheeltool_left\WObj:=Workobject_1;
        MoveJ Target_70,v1000,z0,wheeltool_left\WObj:=Workobject_1;
        MoveJ Target_80,v1000,z0,wheeltool_left\WObj:=Workobject_1;
        MoveJ Target_100,v1000,z0,wheeltool_left\WObj:=Workobject_1;
        MoveL Target_90,v1000,fine,wheeltool_left\WObj:=Workobject_1;
        WaitTime 1;
        SetDO doGrippedLeftWheel, 0;
        WaitTime 1;
        MoveJ Target_80,v1000,z0,wheeltool_left\WObj:=Workobject_1;
        SetDO doStartBelt, 1;
    ENDPROC
ENDMODULE

--- Backups/Controller23/RAPID/TASK2/PROGMOD/CalibData.mod ---
MODULE CalibData
    PERS tooldata wheeltool_right:=[TRUE,[[0,0,20],[1,0,0,0]],[1,[0,0,1],[1,0,0,0],0,0,0]];
    TASK PERS wobjdata Workobject_3:=[FALSE,TRUE,"",[[-358.75,-4997.47,-123.444],[0,1,0,0]],[[0,0,0],[1,0,0,0]]];
    PERS tooldata wheeltool:=[TRUE,[[0,0,20],[1,0,0,0]],[1,[0,0,1],[1,0,0,0],0,0,0]];
ENDMODULE

--- Backups/Controller23/RAPID/TASK2/PROGMOD/Module1.mod ---
MODULE Module1
    CONST robtarget Target_30:=[[1541.158637195,-1119.359435559,-1763.444],[0,0.5,0,0.866025404],[-1,0,-1,0],[0,9E+09,9E+09,9E+09,9E+09,9E+09]];
    CONST robtarget Target_20:=[[477.708443294,360.814777373,-1009.865826741],[0.521902544,-0.125506795,-0.250280456,-0.80574529],[-1,-1,0,0],[0,9E+09,9E+09,9E+09,9E+09,9E+09]];
    CONST robtarget Target_10_2:=[[520.671,400.592,-253.471],[1,0,0,0],[-1,0,1,0],[0,9E+09,9E+09,9E+09,9E+09,9E+09]];
    CONST robtarget Target_10:=[[520.671,400.592,-153.471],[1,0,0,0],[-1,0,1,0],[0,9E+09,9E+09,9E+09,9E+09,9E+09]];
    CONST robtarget Target_40:=[[274.74333609,-2205.172082905,-1332.675203529],[0.688038778,0.210987533,-0.220490433,0.658385047],[1,0,-1,0],[0,9E+09,9E+09,9E+09,9E+09,9E+09]];
    CONST robtarget Target_50:=[[369.43,-2251.172,-314.222],[0.5,0.5,0.5,-0.5],[0,-3,-1,0],[0,9E+09,9E+09,9E+09,9E+09,9E+09]];
    CONST robtarget Target_60:=[[3831.345553083,-1119.359435559,-1763.444],[0,0.5,0,0.866025404],[-1,0,-1,0],[2290.186915888,9E+09,9E+09,9E+09,9E+09,9E+09]];
    CONST robtarget Target_70:=[[2461.119845539,89.729943109,-1763.444],[0.64936295,-0.330821079,-0.374909874,-0.572998917],[-2,-1,0,0],[2290.186915888,9E+09,9E+09,9E+09,9E+09,9E+09]];
    CONST robtarget Target_80_2:=[[2503.123,511.716,-373.3],[1,0,0,0],[-2,0,0,0],[2290.186915888,9E+09,9E+09,9E+09,9E+09,9E+09]];
    CONST robtarget Target_80:=[[2503.123,511.716,-273.3],[1,0,0,0],[-2,0,0,0],[2290.186915888,9E+09,9E+09,9E+09,9E+09,9E+09]];
    CONST robtarget Target_90:=[[1524.20569209,-2336.741920845,-1763.444],[0.625707634,0.345682878,-0.361252471,0.598740308],[1,0,-1,0],[1300.934579439,9E+09,9E+09,9E+09,9E+09,9E+09]];
    CONST robtarget Target_100:=[[1433.625266941,-2422.35908581,-403.788120677],[0.5,0.5,0.5,-0.5],[1,-2,-1,0],[1300.934579439,9E+09,9E+09,9E+09,9E+09,9E+09]];
    CONST robtarget Target_50_3:=[[369.43,-2151.172,-314.222],[0.5,0.5,0.5,-0.5],[0,1,-1,0],[0,9E+09,9E+09,9E+09,9E+09,9E+09]];
    CONST robtarget Target_100_2:=[[1548.919,-2262.172,-379.222],[0.5,0.5,0.5,-0.5],[1,-2,0,0],[1300.934579439,9E+09,9E+09,9E+09,9E+09,9E+09]];
    CONST robtarget Target_110:=[[358.855570616,-2406.697778047,-358.757242225],[0.5,0.5,0.5,-0.5],[0,-3,-1,0],[0,9E+09,9E+09,9E+09,9E+09,9E+09]];
    !***********************************************************
    !
    ! Module:  Module1
    !
    ! Description:
    !   <Insert description here>
    !
    ! Author: tmoun
    !
    ! Version: 1.0
    !
    !***********************************************************


    !***********************************************************
    !
    ! Procedure main
    !
    !   This is the entry point of your program
    !
    !***********************************************************
    PROC main()
        !Add your code here
        SetDo doGrippedRightWheel, 0;
        WaitDI diGripWheel,0;
        SetDO doStartBelt, 0;
        WaitTime 10;
        Path_10;
        Path_20;
    ENDPROC
    PROC Path_10()
        SetDO doStartBelt, 0;
        WaitTime 35;
        MoveJ Target_30,v1000,z0,wheeltool_right\WObj:=Workobject_3;
        MoveJ Target_20,v1000,z0,wheeltool_right\WObj:=Workobject_3;
        MoveL Target_10_2,v1000,fine,wheeltool_right\WObj:=Workobject_3;
        MoveL Target_10,v1000,fine,wheeltool_right\WObj:=Workobject_3;
        WaitTime 2;
        SetDo doGrippedRightWheel, 1;
        WaitTime 1;
        MoveL Target_10_2,v1000,fine,wheeltool_right\WObj:=Workobject_3;
        MoveJ Target_20,v1000,z0,wheeltool_right\WObj:=Workobject_3;
        MoveJ Target_30,v1000,z0,wheeltool_right\WObj:=Workobject_3;
        MoveJ Target_40,v1000,z0,wheeltool_right\WObj:=Workobject_3;
        MoveL Target_110,v1000,fine,wheeltool_right\WObj:=Workobject_3;
        WaitTime 1;
        SetDo doGrippedRightWheel, 0;
        WaitTime 1;
        MoveL Target_40,v1000,fine,wheeltool_right\WObj:=Workobject_3;
        MoveL Target_30,v1000,fine,wheeltool_right\WObj:=Workobject_3;
    ENDPROC
    PROC Path_20()
        MoveJ Target_30,v1000,z0,wheeltool_right\WObj:=Workobject_3;
        MoveJ Target_60,v1000,z0,wheeltool_right\WObj:=Workobject_3;
        MoveJ Target_70,v1000,z0,wheeltool_right\WObj:=Workobject_3;
        MoveL Target_80_2,v1000,fine,wheeltool_right\WObj:=Workobject_3;
        MoveL Target_80,v1000,fine,wheeltool_right\WObj:=Workobject_3;
        WaitTime 1;
        SetDo doGrippedRightWheel, 1;
        WaitTime 1;
        MoveL Target_80_2,v1000,fine,wheeltool_right\WObj:=Workobject_3;
        MoveJ Target_70,v1000,z0,wheeltool_right\WObj:=Workobject_3;
        MoveJ Target_90,v1000,z0,wheeltool_right\WObj:=Workobject_3;
        MoveL Target_100,v1000,fine,wheeltool_right\WObj:=Workobject_3;
        WaitTime 1;
        SetDo doGrippedRightWheel, 0;
        WaitTime 1;
        MoveL Target_90,v1000,fine,wheeltool_right\WObj:=Workobject_3;
        MoveJ Target_60,v1000,fine,wheeltool_right\WObj:=Workobject_3;
        SetDO doStartBelt, 1;
    ENDPROC
ENDMODULE

--- Backups/Controller25/RAPID/TASK1/PROGMOD/CalibData.mod ---
MODULE CalibData
    PERS tooldata sideTool:=[TRUE,[[-24.266,86.667,225],[0.680919208,-0.707106781,0,0.19065422]],[1,[0,0,1],[1,0,0,0],0,0,0]];
    TASK PERS wobjdata Workobject_2:=[FALSE,TRUE,"",[[1567.515,-1038.279,435],[0,0.707106781,0.707106781,0]],[[0,0,0],[1,0,0,0]]];
    PERS tooldata hoodWindTool:=[TRUE,[[0,0,160],[1,0,0,0]],[1,[0,0,1],[1,0,0,0],0,0,0]];
    TASK PERS wobjdata Workobject_4:=[FALSE,TRUE,"",[[1169.19,1406.514,435],[0,0,1,0]],[[0,0,0],[1,0,0,0]]];
ENDMODULE

--- Backups/Controller25/RAPID/TASK1/PROGMOD/Module1.mod ---
MODULE Module1
    CONST robtarget Target_40:=[[1038.279,1567.818934699,-1380],[0.612372436,-0.353553391,-0.353553391,-0.612372436],[-1,0,-1,0],[9E+09,9E+09,9E+09,9E+09,9E+09,9E+09]];
    CONST robtarget Target_20:=[[480.154048262,484.441311489,-120.060966033],[0.999790212,0.019659813,0.005723411,0.000516492],[-1,-1,0,0],[9E+09,9E+09,9E+09,9E+09,9E+09,9E+09]];
    CONST robtarget Target_30:=[[577.699850786,1890.312333014,-478.295945109],[0.999999786,0.000654631,0,0],[-1,-1,0,0],[9E+09,9E+09,9E+09,9E+09,9E+09,9E+09]];
    CONST robtarget Target_50:=[[-2304.864799673,-1535.629168945,-600.156765407],[0.833862645,-0.551924048,0.006916908,0.002256457],[-1,2,-3,1],[9E+09,9E+09,9E+09,9E+09,9E+09,9E+09]];
    CONST robtarget Target_20_3:=[[479.007575376,488.371857989,-219.977112897],[0.999790212,0.019659813,0.005723411,0.000516492],[-1,-1,0,0],[9E+09,9E+09,9E+09,9E+09,9E+09,9E+09]];
    CONST robtarget Target_30_2:=[[552.678048262,1909.215147885,-578.295859401],[0.999999786,0.000654631,0,0],[-1,-1,0,0],[9E+09,9E+09,9E+09,9E+09,9E+09,9E+09]];
    CONST robtarget Target_60:=[[-1966.143934699,-1406.514,-1380],[0.866025404,0,-0.5,0],[0,-1,0,0],[9E+09,9E+09,9E+09,9E+09,9E+09,9E+09]];
    CONST robtarget Target_10_2:=[[573.294688511,562.082048262,-130.117],[1,0,0,0],[0,1,-2,1],[9E+09,9E+09,9E+09,9E+09,9E+09,9E+09]];
    CONST robtarget Target_10:=[[573.294688511,562.082048262,-30.117],[1,0,0,0],[0,2,-2,1],[9E+09,9E+09,9E+09,9E+09,9E+09,9E+09]];
    !***********************************************************
    !
    ! Module:  Module1
    !
    ! Description:
    !   <Insert description here>
    !
    ! Author: tmoun
    !
    ! Version: 1.0
    !
    !***********************************************************


    !***********************************************************
    !
    ! Procedure main
    !
    !   This is the entry point of your program
    !
    !***********************************************************
    PROC main()
        !Add your code here
        SetDo doGripWindsheild, 0;
        SetDO doGripHood, 0;
        SetDO doGenerate, 1;
        SetDO doGenerate, 0;
        SetDO doStartBelt, 0;
        WaitTime 5;
        Path_10;
        Path_20;
    ENDPROC
    PROC Path_10()
        WaitTime 15;
        MoveJ Target_40,v1000,z0,hoodWindTool\WObj:=Workobject_2;
        MoveJ Target_20_3,v1000,z0,hoodWindTool\WObj:=Workobject_2;
        MoveL Target_20,v1000,fine,hoodWindTool\WObj:=Workobject_2;
        WaitTime 1;
        SetDO doGripHood, 1;
        WaitTime 1;
        MoveJ Target_30_2,v1000,z0,hoodWindTool\WObj:=Workobject_2;
        MoveL Target_30,v1000,fine,hoodWindTool\WObj:=Workobject_2;
        WaitTime 1;
        SetDO doGripHood, 0;
        WaitTime 1;
         MoveJ Target_40,v1000,z0,hoodWindTool\WObj:=Workobject_2;
    ENDPROC
    PROC Path_20()
        SetDO doStartBelt, 0;
        WaitTime 5;
        MoveJ Target_60,v1000,z0,hoodWindTool\WObj:=Workobject_4;
        MoveJ Target_10_2,v1000,z0,hoodWindTool\WObj:=Workobject_4;
        MoveL Target_10,v1000,fine,hoodWindTool\WObj:=Workobject_4;
        WaitTime 1;
        SetDo doGripWindsheild, 1;
        WaitTime 1;
        MoveL Target_50,v1000,fine,hoodWindTool\WObj:=Workobject_4;
        WaitTime 1;
        SetDo doGripWindsheild, 0;
        WaitTime 1;
        MoveJ Target_60,v1000,z0,hoodWindTool\WObj:=Workobject_4;
        SetDO doStartBelt, 1;
    ENDPROC
ENDMODULE

--- Backups/Controller25/RAPID/TASK2/PROGMOD/CalibData.mod ---
MODULE CalibData
    PERS tooldata sideTool:=[TRUE,[[-24.266,86.667,225],[0.680919208,-0.707106781,0,0.19065422]],[1,[0,0,1],[1,0,0,0],0,0,0]];
    TASK PERS wobjdata Workobject_5:=[FALSE,TRUE,"",[[5484.225,-1002.89,435],[0,0,1,0]],[[0,0,0],[1,0,0,0]]];
    PERS tooldata seatTool:=[TRUE,[[-5.4,0,164.636],[0.999469999,0,-0.032553365,0]],[1,[0,0,1],[1,0,0,0],0,0,0]];
ENDMODULE

--- Backups/Controller25/RAPID/TASK2/PROGMOD/Module1.mod ---
MODULE Module1
    CONST robtarget Target_30:=[[1678.071701975,925.469341705,-1382.35853718],[0,0.52792704,0,0.849289727],[0,-1,0,0],[9E+09,9E+09,9E+09,9E+09,9E+09,9E+09]];
    CONST robtarget Target_40:=[[347.860688511,1249.696048262,-48.907],[0.54296033,-0.316160544,0.60331347,-0.491171505],[-1,0,0,0],[9E+09,9E+09,9E+09,9E+09,9E+09,9E+09]];
    CONST robtarget Target_50:=[[1453.552115271,1131.912758332,-181.720214692],[0.54296033,-0.316160544,0.60331347,-0.491171505],[-1,0,0,0],[9E+09,9E+09,9E+09,9E+09,9E+09,9E+09]];
    CONST robtarget Target_10_2:=[[2019.129688511,1267.412482525,-299.540972298],[0.687654919,-0.164714032,-0.164714032,-0.687654919],[-1,-1,1,0],[9E+09,9E+09,9E+09,9E+09,9E+09,9E+09]];
    CONST robtarget Target_10:=[[2019.129688511,1312.719048262,-210.393257234],[0.687654919,-0.164714032,-0.164714032,-0.687654919],[-1,-1,1,0],[9E+09,9E+09,9E+09,9E+09,9E+09,9E+09]];
    CONST robtarget Target_20_2:=[[513.259688511,275.460873524,-213.276359217],[0.678863147,-0.197850517,-0.197850517,-0.678863147],[0,-1,1,0],[9E+09,9E+09,9E+09,9E+09,9E+09,9E+09]];
    CONST robtarget Target_20:=[[513.259688511,329.186243428,-128.934290066],[0.678863147,-0.197850517,-0.197850517,-0.678863147],[0,-1,1,0],[9E+09,9E+09,9E+09,9E+09,9E+09,9E+09]];
    !***********************************************************
    !
    ! Module:  Module1
    !
    ! Description:
    !   <Insert description here>
    !
    ! Author: tmoun
    !
    ! Version: 1.0
    !
    !***********************************************************


    !***********************************************************
    !
    ! Procedure main
    !
    !   This is the entry point of your program
    !
    !***********************************************************
    PROC main()
        !Add your code here

        SetDO doGripSeat, 0;
        SetDO doGenerate, 1;
        SetDO doGenerate, 0;

        WaitTime 5;
        Path_10;
    ENDPROC
    PROC Path_10()
        WaitTime 15;
        MoveJ Target_30,v1000,z0,seatTool\WObj:=Workobject_5;
        MoveJ Target_20_2,v1000,z0,seatTool\WObj:=Workobject_5;
        MoveL Target_20,v1000,fine,seatTool\WObj:=Workobject_5;
        WaitTime 1;
        SetDO doGripSeat, 1;
        WaitTime 1;
        MoveJ Target_10_2,v1000,z0,seatTool\WObj:=Workobject_5;
        MoveL Target_10,v1000,fine,seatTool\WObj:=Workobject_5;
        WaitTime 1;
        SetDO doGripSeat, 0;
        WaitTime 1;
        MoveJ Target_30,v1000,z0,seatTool\WObj:=Workobject_5;
    ENDPROC
ENDMODULE

--- Backups/Controller29/RAPID/TASK1/PROGMOD/CalibData.mod ---
MODULE CalibData
    PERS tooldata seatTool:=[TRUE,[[-5.4,0,164.636],[0.99947,0,-0.0325534,0]],[1,[0,0,1],[1,0,0,0],0,0,0]];
    PERS tooldata sideTool:=[TRUE,[[-24.266,86.667,225],[0.680919,-0.707107,0,0.190654]],[1,[0,0,1],[1,0,0,0],0,0,0]];
    TASK PERS wobjdata Workobject_4:=[FALSE,TRUE,"",[[992.538,-209.548,471.4],[0,0.707107,0.707107,0]],[[0,0,0],[1,0,0,0]]];
ENDMODULE

--- Backups/Controller29/RAPID/TASK1/PROGMOD/Module1.mod ---
MODULE Module1
    CONST robtarget Target_30:=[[296.215,415.694272381,-1087.114972448],[0.283727543,-0.741160443,0.259677853,-0.550224765],[0,-1,0,0],[9E+09,9E+09,9E+09,9E+09,9E+09,9E+09]];
    CONST robtarget Target_10_2:=[[269.858922705,465.010889932,-333.14],[0.160293487,0,0,-0.987069399],[0,0,-2,0],[9E+09,9E+09,9E+09,9E+09,9E+09,9E+09]];
    CONST robtarget Target_10:=[[269.858922705,465.010889932,-183.14],[0.160293487,0,0,-0.987069399],[0,0,-2,0],[9E+09,9E+09,9E+09,9E+09,9E+09,9E+09]];
    CONST robtarget Target_20_2:=[[-809.903077295,14.344889932,-524.330266164],[0.776954151,0,0,-0.629557183],[-1,0,-2,0],[9E+09,9E+09,9E+09,9E+09,9E+09,9E+09]];
    CONST robtarget Target_20:=[[-809.903077295,14.344889932,-424.330266164],[0.776954151,0,0,-0.629557183],[-1,0,-2,0],[9E+09,9E+09,9E+09,9E+09,9E+09,9E+09]];
    CONST robtarget Target_40:=[[1263.013922705,401.436889932,-76.585],[0.707106657,-0.67657955,0.000418807,0.205523996],[0,0,1,0],[9E+09,9E+09,9E+09,9E+09,9E+09,9E+09]];
    CONST robtarget Target_50:=[[-873.989388915,442.854728391,-250.069909858],[0.370964602,-0.46436458,-0.468108764,0.653930414],[-1,0,1,0],[9E+09,9E+09,9E+09,9E+09,9E+09,9E+09]];
    CONST robtarget Target_40_2:=[[1290.765361002,305.736894213,-85.032987441],[0.707106657,-0.67657955,0.000418807,0.205523996],[0,-1,0,0],[9E+09,9E+09,9E+09,9E+09,9E+09,9E+09]];
    !***********************************************************
    !
    ! Module:  Module1
    !
    ! Description:
    !   <Insert description here>
    !
    ! Author: tmoun
    !
    ! Version: 1.0
    !
    !***********************************************************


    !***********************************************************
    !
    ! Procedure main
    !
    !   This is the entry point of your program
    !
    !***********************************************************
    PROC main()
        !Add your code here
        SetDO doGenerate,1;
        SetDO doGenerate,0;
        SetDO doStartBelt,1;
        SetDO doGrippedLeftside, 0;
        WaitDI diGripSide,0;
        WaitTime 5;
        Path_10;

    ENDPROC
    PROC Path_10()
        MoveJ Target_30,v1000,z0,sideTool\WObj:=Workobject_4;
        MoveJ Target_40_2,v1000,z0,sideTool\WObj:=Workobject_4;
        MoveL Target_40,v1000,fine,sideTool\WObj:=Workobject_4;
        WaitTime 1;
        SetDO doGrippedLeftside, 1;
        WaitTime 1;
        MoveL Target_50,v1000,fine,sideTool\WObj:=Workobject_4;
        WaitTime 1;
        SetDO doGrippedLeftside, 0;
        WaitTime 1;
        MoveJ Target_30,v1000,z0,sideTool\WObj:=Workobject_4;
    ENDPROC
ENDMODULE

--- Backups/Controller29/RAPID/TASK2/PROGMOD/CalibData.mod ---
MODULE CalibData
    PERS tooldata sideTool:=[TRUE,[[-24.266,86.667,225],[0.680919,-0.707107,0,0.190654]],[1,[0,0,1],[1,0,0,0],0,0,0]];
    TASK PERS wobjdata Workobject_1:=[FALSE,TRUE,"",[[992.538,-209.548,471.4],[0,0.707107,0.707107,0]],[[0,0,0],[1,0,0,0]]];
    PERS tooldata hoodWindTool:=[TRUE,[[0,0,160],[1,0,0,0]],[1,[0,0,1],[1,0,0,0],0,0,0]];
    TASK PERS wobjdata Workobject_2:=[FALSE,TRUE,"",[[1190.48,-2992.07,435],[0,1,-0.000037383,0]],[[0,0,0],[1,0,0,0]]];
ENDMODULE

--- Backups/Controller29/RAPID/TASK2/PROGMOD/Module1.mod ---
MODULE Module1
    CONST robtarget Target_10:=[[360.288165202,1285.471143635,-149.63118002],[0.496895586,-0.35934575,0.586841942,-0.528755088],[-1,-1,0,0],[9E+09,9E+09,9E+09,9E+09,9E+09,9E+09]];
    CONST robtarget Target_30:=[[233.071302161,173.947116952,-1123.514972448],[0.188464037,0.340433148,-0.707712273,0.589686287],[0,-1,0,0],[9E+09,9E+09,9E+09,9E+09,9E+09,9E+09]];
    CONST robtarget Target_10_3:=[[275.550363829,1309.451299081,-67.811433367],[0.503332873,-0.366504615,0.582397802,-0.522631022],[-1,-1,0,0],[9E+09,9E+09,9E+09,9E+09,9E+09,9E+09]];
    CONST robtarget Target_20:=[[291.329148069,-835.062281254,-229.668349884],[0.012258989,0.227678572,0.784230062,-0.577057533],[0,0,-1,0],[9E+09,9E+09,9E+09,9E+09,9E+09,9E+09]];
    CONST robtarget Target_40:=[[355.477065976,1285.472503289,-75.96754803],[0.462818306,-0.380554206,0.655854692,-0.459164823],[-1,0,0,0],[9E+09,9E+09,9E+09,9E+09,9E+09,9E+09]];
    CONST robtarget Target_40_2:=[[164.165601062,1335.479683541,-45.980795688],[0.462818306,-0.380554206,0.655854692,-0.459164823],[-1,0,0,0],[9E+09,9E+09,9E+09,9E+09,9E+09,9E+09]];
    !***********************************************************
    !
    ! Module:  Module1
    !
    ! Description:
    !   <Insert description here>
    !
    ! Author: tmoun
    !
    ! Version: 1.0
    !
    !***********************************************************


    !***********************************************************
    !
    ! Procedure main
    !
    !   This is the entry point of your program
    !
    !***********************************************************
    PROC main()
        !Add your code here
        SetDO doGenerate,1;
        SetDO doGenerate,0;
        SetDO doStartBelt,1;
        SetDO doGrippedRightside, 0;
        WaitDI diGripSide,0;
        WaitTime 5;
        Path_10;
    ENDPROC
    PROC Path_10()
        SetDO doStartBelt, 0;
        MoveJ Target_30,v1000,z0,sideTool\WObj:=Workobject_2;
        MoveJ Target_40_2,v1000,z0,sideTool\WObj:=Workobject_2;
        MoveL Target_40,v1000,fine,sideTool\WObj:=Workobject_2;
        WaitTime 1;
        SetDO doGrippedRightside, 1;
        WaitTime 1;
        MoveL Target_20,v1000,fine,sideTool\WObj:=Workobject_2;
        WaitTime 1;
        SetDO doGrippedRightside, 0;
        WaitTime 1;
        MoveJ Target_30,v1000,z0,sideTool\WObj:=Workobject_2;
        WaitTime 2;
        SetDO doStartBelt, 1;
    ENDPROC
ENDMODULE

--- Backups/Controller23/SYSPAR/EIO.cfg ---
EIO:CFG_1.0:6:1::
#
INDUSTRIAL_NETWORK:

      -Name "PROFIBUS" -Label "PROFIBUS Controller Network"\
      -CfgPath "HOME/pbus_cfg.bin"
#
PROFIBUS_DEVICE:

      -Name "Board10"
#
EIO_SIGNAL:

      -Name "diGripWheel" -SignalType "DI" -Device "Board10" -DeviceMap "0"

      -Name "doGrippedLeftWheel" -SignalType "DO" -Device "Board10"\
      -DeviceMap "1"

      -Name "doGenerateTyre" -SignalType "DO" -Device "Board10" -DeviceMap "2"

      -Name "doGrippedRightWheel" -SignalType "DO" -Device "Board10"\
      -DeviceMap "3"

      -Name "doStartBelt" -SignalType "DO" -Device "Board10" -DeviceMap "4"

--- Backups/Controller25/SYSPAR/EIO.cfg ---
EIO:CFG_1.0:6:1::
#
INDUSTRIAL_NETWORK:

      -Name "PROFIBUS" -Label "PROFIBUS Controller Network"\
      -CfgPath "HOME/pbus_cfg.bin"
#
PROFIBUS_DEVICE:

      -Name "Board10"
#
EIO_SIGNAL:

      -Name "diStart" -SignalType "DI" -Device "Board10" -DeviceMap "0"

      -Name "doGripSeat" -SignalType "DO" -Device "Board10" -DeviceMap "1"

      -Name "doGripHood" -SignalType "DO" -Device "Board10" -DeviceMap "2"

      -Name "doGenerate" -SignalType "DO" -Device "Board10" -DeviceMap "3"

      -Name "doGripWindsheild" -SignalType "DO" -Device "Board10" -DeviceMap "4"

      -Name "doStartBelt" -SignalType "DO" -Device "Board10" -DeviceMap "5"

--- Backups/Controller29/SYSPAR/EIO.cfg ---
EIO:CFG_1.0:6:1::
#
INDUSTRIAL_NETWORK:

      -Name "PROFIBUS" -Label "PROFIBUS Controller Network"\
      -CfgPath "HOME/pbus_cfg.bin"
#
PROFIBUS_DEVICE:

      -Name "Board10"
#
EIO_SIGNAL:

      -Name "doGenerate" -SignalType "DO" -Device "Board10" -DeviceMap "0"

      -Name "doStartBelt" -SignalType "DO" -Device "Board10" -DeviceMap "1"

      -Name "distartbelt" -SignalType "DI" -Device "Board10" -DeviceMap "2"

      -Name "diGripSide" -SignalType "DI" -Device "Board10" -DeviceMap "3"

      -Name "doGrippedLeftside" -SignalType "DO" -Device "Board10"\
      -DeviceMap "4"

      -Name "doGrippedRightside" -SignalType "DO" -Device "Board10"\
      -DeviceMap "5"
